{attribute 'qualified_only'}
{attribute 'strict'}
{attribute 'to_string'}
TYPE E_VacuumzuignapStatus :
(
	SturingVacuumLoslaten := 0,
	SturingVacuumOpppakken
);
END_TYPE

(* stored: Version 1.1.0.1
   DUT E_VacuumzuignapStatus: Id {d6269f93-2033-4cdf-8883-5f78d3f4a092} *)
